Fanuc TP program (LS listing): _fence.ls

/PROG  _FENCE	  Cond
/ATTR
OWNER		= MNEDITOR;
COMMENT		= "";
PROG_SIZE	= 191;
CREATE		= DATE 21-08-19  TIME 21:16:04;
MODIFIED	= DATE 21-08-19  TIME 21:16:04;
FILE_NAME	= ;
VERSION		= 0;
LINE_COUNT	= 1;
MEMORY_SIZE	= 567;
PROTECT		= READ_WRITE;
TCD:  STACK_SIZE	= 0,
      TASK_PRIORITY	= 50,
      TIME_SLICE	= 0,
      BUSY_LAMP_OFF	= 0,
      ABORT_REQUEST	= 7,
      PAUSE_REQUEST	= 7;
DEFAULT_GROUP	= *,*,*,*,*;
CONTROL_CODE	= 00000000 00000000;
/APPL
/APPL

AUTO_SINGULARITY_HEADER;
  ENABLE_SINGULARITY_AVOIDANCE   : TRUE;
/MN
   1:  WHEN DO[119]=ON,CALL ABORTALL ;
/POS
/END
